PROGRAM MAIN

// Blowfish test
P_Blowfish();

END_PROGRAM

(* stored: Version 1.1.0.1, ProductVersion 3.1.4024.9
   POU MAIN: Id {5ede9854-04af-4c4d-b59a-9eb30d0070e2}, SpecialFunc None *)
